{attribute 'linkalways'} 
{attribute 'no_explicit_call' := 'This FB is a CLASS and must be accessed using methods or properties'}
{attribute 'enable_dynamic_creation'}
FUNCTION_BLOCK SafeMemCopyOperation EXTENDS Disposable IMPLEMENTS I_DatatypeOperation
VAR
	source : I_Datatype;
	destination : I_Datatype;
END_VAR

METHOD Execute
VAR
END_VAR
destination.TryCopyFrom(source);
END_METHOD

METHOD FB_init : BOOL
VAR_INPUT
	bInitRetains : BOOL; // if TRUE, the retain variables are initialized (warm start / cold start)
	bInCopyCode : BOOL;  // if TRUE, the instance afterwards gets moved into the copy code (online change)
	Source : I_Datatype;
	Destination : I_Datatype;
END_VAR
THIS^.source := Source;
This^.destination := Destination;
END_METHOD

END_FUNCTION_BLOCK

(* stored: Version 1.1.0.1, ProductVersion 3.1.4024.12
   POU SafeMemCopyOperation: Id {3fc77062-f732-474c-a8ea-007ea8126945}, SpecialFunc None
   Folder Constructor: Id {2f0874a3-84d5-4ec9-9ae1-badd817e47a9}
   Method Execute: Id {aa4b5bd4-b214-4709-a00d-aae796131268}
   Method FB_init: Id {42940293-215f-4a4e-8899-0f68e0cff581} *)
